FUNCTION_BLOCK EmptySimple (* Template for an empty simple function block *)
  (* Standard: 61499-1 *)
  (* Version 0.0, 2018-10-15, Peter Gsellmann, TU Wien/ACIN *)
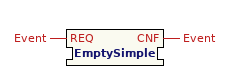
  EVENT_INPUT
    REQ; (* Normal Execution Request *)
  END_EVENT
  EVENT_OUTPUT
    CNF; (* Execution Confirmation *)
  END_EVENT
  ALGORITHM REQ IN AnyText:

  END_ALGORITHM
END_FUNCTION_BLOCK
